FUNCTION_BLOCK Stage3 (* Template for a Basic Function Block Type *)
  (* Standard: 61499-2 *)
  (* Version 1.0, 2021-06-20, HP *)
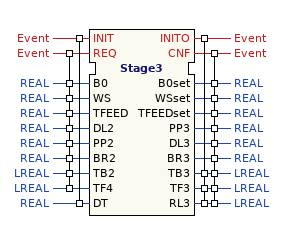
  EVENT_INPUT
    INIT WITH DT; (* Initialization Request *)
    REQ WITH B0, WS, TFEED, DL2, PP2, BR2, TB2, TF4; (* Normal Execution Request *)
  END_EVENT
  EVENT_OUTPUT
    INITO WITH RL3, TF3, TB3; (* Initialization Confirm *)
    CNF WITH PP3, B0set, WSset, TFEEDset, DL3, BR3, TB3, TF3, RL3; (* Execution Confirmation *)
  END_EVENT
  VAR_INPUT
    B0 : REAL;
    WS : REAL;
    TFEED : REAL;
    DL2 : REAL;
    PP2 : REAL;
    BR2 : REAL;
    TB2 : LREAL;
    TF4 : LREAL;
    DT : REAL;
  END_VAR
  VAR_OUTPUT
    B0set : REAL;
    WSset : REAL;
    TFEEDset : REAL;
    PP3 : REAL;
    DL3 : REAL;
    BR3 : REAL;
    TB3 : LREAL;
    TF3 : LREAL;
    RL3 : LREAL;
  END_VAR
  VAR
    AB : REAL; (* internal variabel *)
    UU : REAL;
    TREF : REAL;
    AD : REAL;
    AHC : REAL;
    AHR : REAL;
    AS : REAL;
    REC : REAL;
    WN : REAL;
    WN_1 : REAL;
    XKN : REAL;
    C1 : REAL;
    HS : REAL;
    G : REAL;
    W1 : REAL;
    TFREC : REAL;
    TS : REAL;
    DTS : REAL;
    TF3_last : REAL;
    RL3_last : REAL;
    TB3_last : REAL;
    USS : REAL;
    RHOB : REAL;
    CPB : REAL;
    CPF : REAL;
    FMW : REAL;
    HLV : REAL;
    HV : REAL;
    BPR : REAL;
    FMC : REAL;
    U : REAL;
    A : REAL;
    B : REAL;
    C : REAL;
    D1 : REAL;
    d : REAL;
    a : REAL;
    A1 : REAL;
    A2 : REAL;
    A3 : REAL;
    A4 : REAL;
    A5 : REAL;
    A6 : REAL;
    p : REAL;
    q : REAL;
    TC : REAL;
    PC : REAL;
    DTB3 : REAL;
    DEN3 : REAL;
    DH3 : REAL;
    DP3 : REAL;
    DPDH3 : REAL;
    DT3 : REAL;
    m : REAL;
    n : REAL;
    VR3 : REAL;
    DELTA3 : REAL;
    DELTA25 : REAL;
    DELTA47 : REAL;
    DELTA3_last : REAL;
    DELTA25_last : REAL;
    DELTA47_last : REAL;
  END_VAR
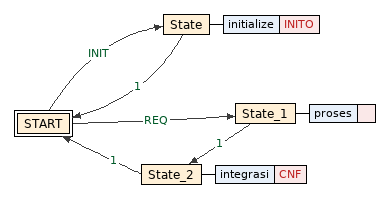
  EC_STATES
    START; (* Initial State *)
    State : initialize -> INITO;
    State_1 : proses;
    State_2 : integrasi -> CNF;
  END_STATES
  EC_TRANSITIONS
    START TO State := INIT;
    State TO START := 1;
    START TO State_1 := REQ;
    State_1 TO State_2 := 1;
    State_2 TO START := 1;
  END_TRANSITIONS
  ALGORITHM initialize IN ST: (* Initialization algorithm *)
TREF :=273.15;
AB :=57.2727;
AHC :=4069.2;
AHR :=2639.7;
AS :=3225.7;
REC :=0.0;
//TF2:=TF2;

//TFEED :=TFEED1+TREF;
 //TS:=TS1+TREF;
WN :=3.0;
XKN :=0.68;
HS:=0.11;
G :=9.81;
W1 :=0.50;

RL3 :=0.528750190123305;
TB3 :=361.282649739703;
TF3 := 354.946694895621;
TF4 := 352.376032234529;


RL3_last :=RL3;
TB3_last :=TB3;
TF3_last :=TF3;
  END_ALGORITHM
  ALGORITHM proses IN ST: (* kalkulasi *)
UU := TFEED;
U :=UU;

USS :=49.767;
C1 :=0.625;
RHOB :=1032.4; //maassa jenis brine
CPB :=1.00; //heatcapacity Brine
CPF :=1.00; //heat capacity feed
FMW :=23654.0;
HLV :=563.7959;
HV :=625.1971;
BPR :=2.192;
FMC :=34736.09;
//U :=UU; //feed temp



///  Calculate the physical properties

//A :=3.2437814;
//B :=5.86826*0.001;
//C :=1.1702379*0.00000001;
//D1 :=2.1878462*0.001;
//TC :=647.27;
//PC :=218.167;


A1 :=3.2437814;
A2:=5.86826*0.001;
A3:=1.1702379*0.00000001;
A4 :=2.1878462*0.001;
A5 :=647.27;
A6 :=218.167;

DTB3 :=A5-TB3;
DEN3 :=(A1+A2*DTB3+A3*DTB3*DTB3*DTB3)/(1+A4*DTB3)*DTB3/TB3;
p:=DEN3;
q:=10.0;
PP3 :=A6/(EXPT(q, p));

// calculate the brine flow rates
DP3:=PP2-PP3;
DH3:=RL3-C1*HS;
DPDH3 :=DP3*101000+G*RHOB*DH3;
m:=DPDH3*RHOB;
n:=0.5;
BR3 :=WN*XKN*RL3*(EXPT(m, n));
BR3 :=BR3*60.0/1000.0;

// calculate the vapor flow rates

DT3 :=TB3-BPR/1.8-(TF4+TF3)*0.5;
VR3 :=U*AHC*DT3/HLV/1000.0;
DL3 :=DL2+VR3;


//// state equation
DELTA3 :=(BR2-BR3-VR3)*1000.0/RHOB/AB;
DELTA25 :=((BR2*CPB*(TB2-TB3))-VR3*(HV-CPB*(TB3-TREF)))*1000.0/AB/RHOB/CPB/RL3;
DELTA47 :=((B0*CPF*(TF4-TF3)*1000+(U*AHC*DT3)))/FMW/CPF;
  END_ALGORITHM
  ALGORITHM integrasi IN ST: (* new algorithm *)
B0set:=B0;
WSset:=WS ;
TFEEDset:=TFEED;
//integrasi
RL3 := (DELTA3 + DELTA3_last)*0.5*DT + RL3_last;
DELTA3_last :=DELTA3 ;
RL3_last :=RL3;

TB3 := (DELTA25 + DELTA25_last)*0.5*DT + TB3_last;
DELTA25_last :=DELTA25 ;
TB3_last:=TB3;

TF3 := (DELTA47 + DELTA47_last)*0.5*DT + TF3_last;
DELTA47_last :=DELTA47 ;
TF3_last :=TF3;
  END_ALGORITHM
END_FUNCTION_BLOCK
